PROGRAM MAIN
VAR

State: Step;

StopButton AT %I*: BOOL;

TimerMotorStart: TON;
TimerPick: TON;
TimerRelease: TON;
TimerZUp: TON;
TimerTrayMotor: TON;
TimerWaitBeforeMove: TON;
	
Xas: AXIS_REF;
Yas: AXIS_REF;
Tray: AXIS_REF;

XMotorPower: MC_power; 
YMotorPower: MC_power;
TrayMotorPower: MC_power;

XMotorPosition: MC_MoveAbsolute;
YMotorPosition: MC_MoveAbsolute;
TrayMotorPosition: MC_MoveAbsolute;

XMotorHome: MC_Home;
YMotorHome: MC_Home;
TrayMotorHome: MC_Home;

XMotorReset: MC_Reset;
YMotorReset: MC_Reset;
TrayMotorReset: MC_Reset;

XMotorJog: MC_Jog;
YMotorJog: MC_Jog;

XJogForward : BOOL;
XJogBackwards : BOOL;

YJogForward : BOOL;
YJogBackwards : BOOL;
 

HomingDone: BOOL;

GripperSmall AT %Q*: BOOL;
GripperWide AT %Q*: BOOL;
Z_Down AT %Q*: BOOL;
Z_Up  AT %Q*: BOOL;
TrayFix_In  AT %Q*: BOOL;
TrayFix_Out  AT %Q*: BOOL;
Vacuum AT %Q*: BOOL;





PodSensor AT %I*: BOOL;



XDefault: INT := 0; 		//Positie van X-as waar de gantry wacht om te picken.
YDefault: INT := 340;		//Positie van Y-as waar de gantry wacht om te picken.


XMove: INT := -8000; //AANVULLEN
YMove: INT := 6125; //AANVULLEN 


DefaultCoordinate: INT := -9395; //AANVULLEN
Coordinate: INT := -9395; //AAMVULLEN		//Variabele voor de huidige rij in de bak.
PlusCoordinate: INT := 946; //AANVULLEN 	
MaxCoordinate: INT := -731 ; //AANVULLEN		//Variabele voor de laatste rij in de bak.


TrayPositionBlock: INT := 180; //AANVULLEN
TrayPositionFree: INT := 0; //AANVULLEN

PickTime: TIME:= T#3S; // TIJD CHECKEN
ReleaseTime: TIME := T#1S; // TIJD CHECKEN
ZUpTime: TIME := T#3S; // TIJD CHECKEN
TrayTime: TIME := T#5S; //TIJD CHECKEN
WaitMoveTime: TIME := T#3990MS; //TIJD CHECKEN
END_VAR

XMotorPosition(Axis := Xas, Velocity := 1333, Acceleration := 2000, Deceleration := 2000, Jerk := 100000);
YMotorPosition(Axis := Yas, Velocity := 1333, Acceleration := 2000, Deceleration := 2000, Jerk := 100000);
TrayMotorPosition(Axis := Tray, Velocity := 90, Acceleration := 180, Deceleration := 180, Jerk := 100000);


CASE State OF
	
Step.IDLE:	

	IO.lamp_geel := FALSE;
	Z_Up := TRUE;
	Z_Down := FALSE;	
	GripperSmall := TRUE;
	GripperWide := FALSE;
	IO.PLC_Ready := TRUE;
	XMotorReset(Axis := XAs, Execute := FALSE);
	YMotorReset(Axis := YAs, Execute := FALSE);
	TrayMotorReset(Axis := Tray, Execute := FALSE);

	

	
	IF NOT IO.EmergencyStop THEN
		State := Step.STOPPED;
	END_IF
	
	
	IF IO.StartButton THEN
			State := Step.STARTING;
	END_IF
			 
		

Step.STARTING:

	XMotorPower(Axis:= Xas, Enable := TRUE, Enable_Positive := TRUE, Enable_Negative := TRUE);
	YMotorPower(Axis:= Yas, Enable := TRUE, Enable_Positive := TRUE, Enable_Negative := TRUE);
	TrayMotorPower(Axis:= Tray, Enable := TRUE, Enable_Positive := TRUE, Enable_Negative := TRUE);	
	IO.lamp_geel := TRUE;
	IO.lamp_groen := FALSE;
	IO.lamp_rood := FALSE;
	TimerMotorStart(IN := TRUE, PT := T#1S);
	
	IF NOT IO.TraySensor AND HomingDone AND NOT TrayMotorPosition.Done THEN
		IO.TrayRequest := TRUE; // Signaal sturen naar AMR.
		TrayFix_Out := FALSE;
		TrayFix_In := TRUE;
	END_IF 	
		
	IF IO.TraySensor AND HomingDone THEN
		TimerTrayMotor(IN := TRUE, PT := TrayTime);
	END_IF
	
	IF TimerTrayMotor.Q THEN
		IO.TrayRequest := FALSE; //Signaal sturen naar AMR.		
		TrayMotorPosition(Axis := Tray, Execute := TRUE, Position := TrayPositionBlock);		
	END_IF
	
	
	IF TrayMotorPosition.Done THEN
		TrayFix_Out := TRUE;
		TrayFix_In := FALSE;
	END_IF
	
	IF NOT IO.EmergencyStop THEN
		State := Step.STOPPED;
	END_IF	
	
	IF NOT HomingDone AND TimerMotorStart.Q THEN
		State := Step.HOMING;
	END_IF	
	
	IF HomingDone AND TimerMotorStart.Q AND IO.TraySensor AND TrayFix_Out AND NOT IO.Trayrequest THEN 
		State := Step.EXECUTE_ZEROING;
	END_IF
	

	
	
Step.HOMING: 

	IF NOT IO.EmergencyStop THEN
		State := Step.STOPPED;
	END_IF
		
	IF IO.StartButton THEN
		IO.HomingSensor := TRUE;
	END_IF
	
	IF IO.HomingSensor = TRUE THEN
		XMotorHome(Axis := Xas, Execute := TRUE, Position := 0, HomingMode := MC_DIRECT);
		YMotorHome(Axis := Yas, Execute := TRUE, Position := 0, HomingMode := MC_DIRECT);
		TrayMotorHome(Axis := Tray, Execute := TRUE, Position := 0, HomingMode := MC_DIRECT);
	END_IF
	IF	XMotorHome.Done AND YMotorHome.Done AND TrayMotorHome.Done THEN
		HomingDone := TRUE;
		State := Step.STARTING;
	END_IF
	
  	
Step.EXECUTE_ZEROING:
	TrayMotorPosition(Axis := Tray, Execute := FALSE);
	IO.lamp_geel := FALSE;
	IO.lamp_groen := TRUE;
	IO.lamp_rood := FALSE;
	XMotorPosition(Axis := Xas, Execute := TRUE, Position := XDefault);
	YMotorPosition(Axis := Yas, Execute := TRUE, Position := YDefault);	
	TimerRelease(IN := FALSE);
	TimerTrayMotor(IN := FALSE);
	TimerZUp(IN := FALSE);
	

	IF NOT IO.EmergencyStop THEN
		State := Step.STOPPED;
	END_IF	
	
	IF  XMotorPosition.Done AND YMotorPosition.Done AND Coordinate < MaxCoordinate AND PodSensor THEN
		XMotorPosition(Axis := Xas, Execute := FALSE);
		YMotorPosition(Axis := Yas, Execute := FALSE);
		State:= Step.EXECUTE_PICK;	
	ELSIF Coordinate > MaxCoordinate THEN
		State:= Step.SUSPENDED;
	END_IF

Step.EXECUTE_PICK:
	GripperSmall := TRUE;
	GripperWide := FALSE;
	TimerWaitBeforeMove(IN := TRUE, PT := WaitMoveTime);
	
	IF NOT IO.EmergencyStop THEN
		State := Step.STOPPED;
	END_IF
	
	IF TimerWaitBeforeMove.Q THEN
		XMotorPosition(Axis := Xas, Execute := TRUE, Position := XMove);
		TimerPick(IN := TRUE, PT := PickTime);
	END_IF
	
	IF TimerPick.Q THEN 
		TimerZUp(IN := TRUE, PT := ZUpTime);
		Z_Up := FALSE;
		Z_Down := TRUE;
		Vacuum := TRUE;
	END_IF
	
	IF  TimerZUp.Q THEN

		Z_Up := TRUE;
		Z_Down := FALSE;						
	END_IF
	
	IF XMotorPosition.Done THEN
		XMotorPosition(Axis := Xas, Execute := FALSE);
		TimerZUp(IN := FALSE);	
 		State := Step.EXECUTE_PLACE;
	END_IF
	
Step.EXECUTE_PLACE:

	TimerPick(IN := FALSE);
	TimerWaitBeforeMove(IN := FALSE);
	
	IF NOT TimerZUp.Q AND NOT TimerPick.Q THEN
		XMotorPosition(Axis := Xas, Execute := TRUE, Position := Coordinate);
		YMotorPosition(Axis := Yas, Execute := TRUE, Position := YMove);
	END_IF
	
	IF Z_Up THEN
		GripperSmall := FALSE;
		GripperWide := TRUE;		
	END_IF
	
	IF NOT IO.EmergencyStop THEN
	State := Step.STOPPED;
	END_IF
	
	IF  XMotorPosition.Done AND YMotorPosition.Done THEN
		Z_Up := FALSE;
		Z_Down := TRUE;	
		TimerRelease(IN := TRUE, PT := ReleaseTime);																
	END_IF
	
	IF TimerRelease.Q THEN
		Vacuum := FALSE;
		TimerZUp(IN := TRUE, PT := ZUpTime);
	END_IF
	
	IF TimerZUp.Q THEN
		Z_Up := TRUE;
		Z_Down := FALSE;
		Coordinate := Coordinate + PlusCoordinate;
		XMotorPosition(Axis := Xas, Execute := FALSE);
		YMotorPosition(Axis := Yas, Execute := FALSE);
		State := Step.EXECUTE_ZEROING;
	END_IF
	

Step.SUSPENDED:
	
	IO.lamp_geel := TRUE;
	IO.lamp_groen := FALSE;
	IO.lamp_rood := FALSE;
	TrayFix_In := TRUE;
	TrayFix_Out := FALSE;
	IO.TrayRequest := TRUE;	
	TrayMotorPosition(Axis := Tray, Execute := TRUE, Position := TrayPositionFree);	
		
	IF NOT IO.TraySensor THEN
		TrayMotorPosition(Axis := Tray, Execute := FALSE);	
		State := Step.UNSUSPENDING;
	END_IF

	IF NOT IO.EmergencyStop THEN
	State := Step.STOPPED;
	END_IF

Step.UNSUSPENDING:

	Coordinate := DefaultCoordinate;
	
	IF IO.TraySensor THEN
		TimerTrayMotor(IN := TRUE, PT := TrayTime);
	END_IF
	
	IF TimerTrayMotor.Q THEN
		TrayMotorPosition(Axis := Tray, Execute := TRUE, Position := TrayPositionBlock);	
	END_IF
	
	IF TrayMotorPosition.Done THEN 
		TrayFix_In := FALSE;
		TrayFix_Out := TRUE;		
		IO.TrayRequest := FALSE;
		State := Step.EXECUTE_ZEROING;
		TimerTrayMotor(IN := FALSE);
	END_IF
	
	IF NOT IO.EmergencyStop THEN
	State := Step.STOPPED;
	END_IF
	
Step.STOPPED:

	IO.lamp_geel := FALSE;
	IO.lamp_groen := FALSE;
	IO.lamp_rood := TRUE;

	TimerMotorStart(IN := FALSE);
	TimerTrayMotor(IN := FALSE);
	XMotorPower(Axis:= Xas, Enable := FALSE, Enable_Positive := FALSE, Enable_Negative := FALSE);
	YMotorPower(Axis:= Yas, Enable := FALSE, Enable_Positive := FALSE, Enable_Negative := FALSE);
	TrayMotorPower(Axis:= Tray, Enable := FALSE, Enable_Positive := FALSE, Enable_Negative := FALSE);
	XMotorPosition(Axis := Xas, Execute := FALSE);
	YMotorPosition(Axis := Yas, Execute := FALSE);
	TrayMotorPosition(Axis := Tray, Execute := FALSE);
	IO.PLC_Ready := FALSE;
	GripperSmall := FALSE;
	GripperWide := FALSE;
	TrayFix_In := FALSE;
	TrayFix_Out := FALSE;
	Z_Down := FALSE;
	Z_Up := FALSE;
	Vacuum := FALSE;
	
	
	IF IO.EmergencyStop AND IO.ResetButton THEN
		State := Step.RESETTING;
	END_IF
	
Step.RESETTING:

	IO.lamp_geel := TRUE;
	IO.lamp_groen := FALSE;
	IO.lamp_rood := FALSE;
	
	IF NOT IO.EmergencyStop THEN
		State := Step.STOPPED;
	END_IF
	
	IF IO.StartButton THEN
		XMotorReset(Axis := XAs, Execute := TRUE);
		YMotorReset(Axis := YAs, Execute := TRUE);
		TrayMotorReset(Axis := Tray, Execute := TRUE);
		State := Step.IDLE;
	END_IF
	

END_CASE

END_PROGRAM

(* stored: Version 1.1.0.1, ProductVersion 3.1.4024.12
   POU MAIN: Id {81c9a74c-03e9-4a27-9583-67c673982615}, SpecialFunc None *)
